FUNCTION_BLOCK E_STOPWATCH (* FB for stopping time between events *)
  (* Standard: 61499-2; Description: Copyright (c) 2018, 2024 fortiss GmbH, Johannes Kepler University Linz, HR Agrartechnik GmbH This program and the accompanying materials are made available under the terms of the Eclipse Public License 2.0 which is available at https://www.eclipse.org/legal/epl-2.0/ SPDX-License-Identifier: EPL-2.0 *)
  (* Version 1.0, 2018-08-29, Ben Schneider, fortiss GmbH, initial API and implementation and/or initial documentation *)
  (* Version 1.1, 2020-05-24, alois Zoitl, Johannes Kepler University Linz, Changed to a full basic FB implementation utilizing the new NOW_MONOTONIC function *)
  (* Version 1.2, 2024-09-19, Franz Höpfinger, HR Agrartechnik GmbH, Added additional Events *)
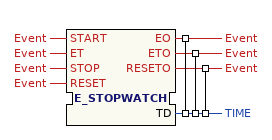
  EVENT_INPUT
    START; (* Start the stopwatch *)
    ET; (* Trigger the Time output *)
    STOP; (* Stop the stopwatch *)
    RESET; (* Reset the stopwatch to 0 *)
  END_EVENT
  EVENT_OUTPUT
    EO WITH TD; (* Event Output *)
    ETO WITH TD; (* Trigger the Time output  confirm *)
    RESETO WITH TD; (* Reset the stopwatch to 0  confirm *)
  END_EVENT
  VAR_OUTPUT
    TD : TIME; (* The measured time difference in milliseconds *)
  END_VAR
  VAR
    startTime : TIME; (* Holds the time value when the start event occured. *)
  END_VAR
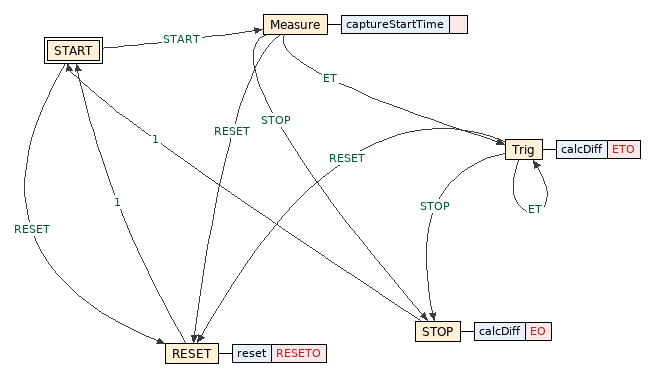
  EC_STATES
    START;
    Measure : captureStartTime;
    STOP : calcDiff -> EO;
    Trig : calcDiff -> ETO;
    RESET : reset -> RESETO;
  END_STATES
  EC_TRANSITIONS
    START TO Measure := START;
    Measure TO STOP := STOP;
    STOP TO START := 1;
    Trig TO STOP := STOP;
    Measure TO Trig := ET;
    Trig TO Trig := ET;
    Measure TO RESET := RESET;
    RESET TO START := 1;
    START TO RESET := RESET;
    Trig TO RESET := RESET;
  END_TRANSITIONS
  ALGORITHM captureStartTime IN ST:
startTime := NOW_MONOTONIC();
  END_ALGORITHM
  ALGORITHM calcDiff IN ST:
TD := NOW_MONOTONIC() - startTime;
  END_ALGORITHM
  ALGORITHM reset IN ST:
TD := T#0s;
  END_ALGORITHM
END_FUNCTION_BLOCK
